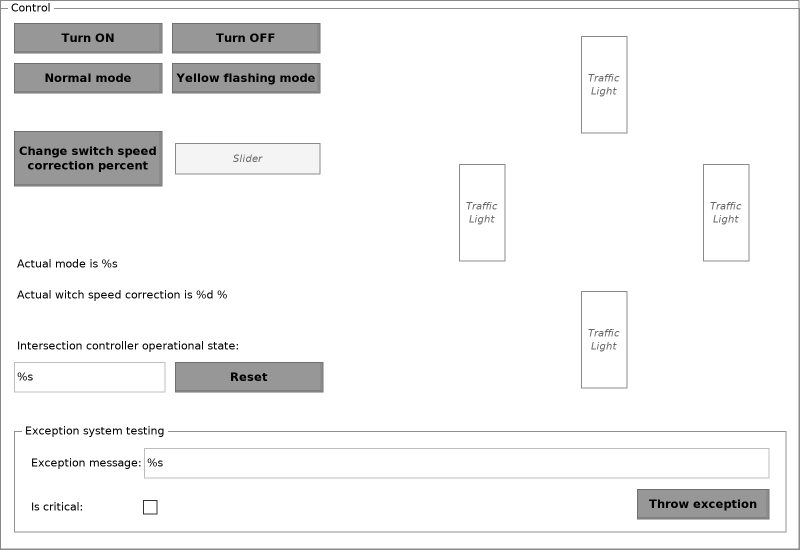
VISUALIZATION Intersection  // 800x550
    GroupBox (0,0 800x550), "Control"
        Rectangle (543,32 120x360), angle 90
        Line (486,126)
        Rectangle (543,24 120x376)
        Frame (581,36 46x97)
            shows TrafficLight(Red := MAIN.IntersectionHMI.TrafficLight2.Statuses.RedLightIsActive, Yellow := MAIN.IntersectionHMI.TrafficLight2.Statuses.YellowLightIsActive, Green := MAIN.IntersectionHMI.TrafficLight2.Statuses.GreenLightIsActive)
        Frame (581,291 46x97)
            shows TrafficLight(Red := MAIN.IntersectionHMI.TrafficLight4.Statuses.RedLightIsActive, Yellow := MAIN.IntersectionHMI.TrafficLight4.Statuses.YellowLightIsActive, Green := MAIN.IntersectionHMI.TrafficLight4.Statuses.GreenLightIsActive)
        Frame (703,164 46x97)
            shows TrafficLight(Red := MAIN.IntersectionHMI.TrafficLight3.Statuses.RedLightIsActive, Yellow := MAIN.IntersectionHMI.TrafficLight3.Statuses.YellowLightIsActive, Green := MAIN.IntersectionHMI.TrafficLight3.Statuses.GreenLightIsActive)
        Frame (459,164 46x97)
            shows TrafficLight(Red := MAIN.IntersectionHMI.TrafficLight1.Statuses.RedLightIsActive, Yellow := MAIN.IntersectionHMI.TrafficLight1.Statuses.YellowLightIsActive, Green := MAIN.IntersectionHMI.TrafficLight1.Statuses.GreenLightIsActive)
        Textfield (14,362 151x30), "%s", text variable: MAIN.IntersectionHMI.AutomationComponentStatuses.OperationalStateName, input disabled if: FALSE
        Label (14,331 270x30), "Intersection controller operational state:"
        Slider (175,143 145x31), variable: MAIN.IntersectionHMI.Commands.SwitchingSpeedCorrectionPercent, scale -30..30
        GroupBox (14,423 772x109), "Exception system testing"
            Label (14,25 116x30), "Exception message:"
            Textfield (130,25 625x30), "%s", text variable: MAIN.IntersectionHMI.Commands.ExceptionMessage, input disabled if: FALSE
                OnMouseClick: write the text variable via Default
            Button (623,66 132x30), "Throw exception"
                OnMouseClick: execute { MAIN.IntersectionHMI.Commands.ThrowExceptionInDemoExceptionGenerator := TRUE; }
            Label (14,68 110x30)
            Label (14,69 110x30), "Is critical:"
            Checkbox (127,69 28x30), variable: MAIN.IntersectionHMI.Commands.ExceptionIsCritical
        Button (175,362 148x30), "Reset"
            OnMouseClick: execute { MAIN.IntersectionHMI.AutomationComponentCommands.Reset := TRUE; }
        Button (14,23 148x30), "Turn ON"
            tap MAIN.IntersectionHMI.Commands.TurnOn
        Button (172,23 148x30), "Turn OFF"
            tap MAIN.IntersectionHMI.Commands.TurnOff
        Button (14,63 148x30), "Normal mode"
            tap MAIN.IntersectionHMI.Commands.SetYellowFlashingModeOff
        Button (172,63 148x30), "Yellow flashing mode"
            tap MAIN.IntersectionHMI.Commands.SetYellowFlashingModeOn
        Button (14,131 148x55), "Change switch speed correction percent"
            tap MAIN.IntersectionHMI.Commands.SetSwitchingSpeedCorrectionPercent
        Textfield (14,249 306x30), "Actual mode is %s", text variable: MAIN.IntersectionHMI.Statuses.ModeName, input disabled if: FALSE
        Textfield (14,280 306x30), "Actual witch speed correction is %d %", text variable: MAIN.IntersectionHMI.Statuses.SwitchingSpeedCorrectionPercent, input disabled if: FALSE
END_VISUALIZATION

(* stored: Version 1.1.0.1
   Visu Intersection: Id {3f36056b-e97d-47c4-837d-733890435638} *)
